PROGRAM main
VAR
	Relay_Start AT %QX4.0 : bool; (* Address modbus: 32 *)
	Start_State AT %QX4.1 : bool; (* Address modbus: 33 *)
	Relay_Downtime AT %QX4.2 : bool; (* Address modbus: 34 *)
	Downtime_State AT %QX4.3 : bool; (* Address modbus: 35 *)
	Counter_Trigger AT %QX4.4 : bool; (* Address modbus: 36 *)
	Reset_Counter AT %QX4.5 : bool; (* Address modbus: 37 *)
	Counter_Register AT %MW10 : int; (* 0 = 1024 --> HR 10 = 1034 *)
	R_TRIG0 : R_TRIG;
	Pulse_Counter : bool;
	CTU0 : CTU;
	R_TRIG1 : R_TRIG;
	Pulse_Reset : bool;
END_VAR

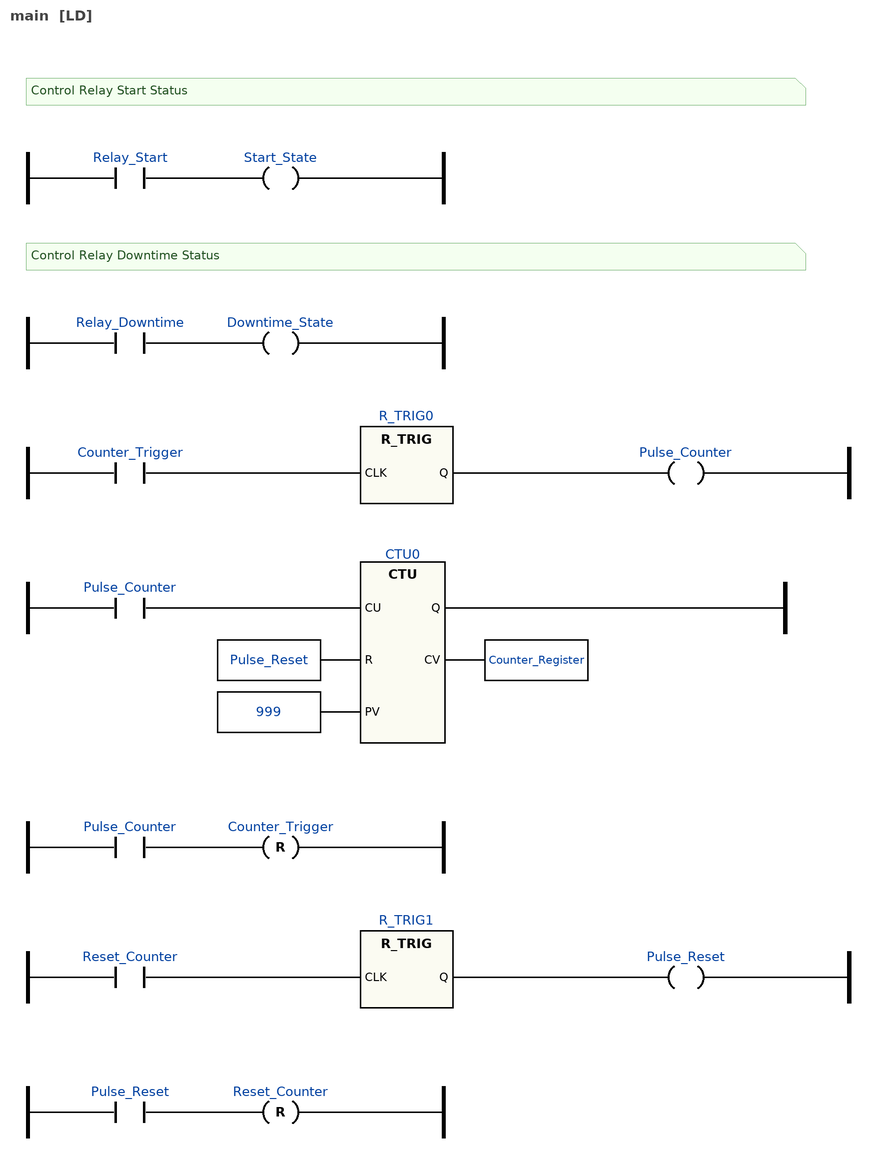
(* LD diagram, written out as Structured Text *)
(* Control Relay Start Status *)
Start_State := Relay_Start;
(* Control Relay Downtime Status *)
Downtime_State := Relay_Downtime;
R_TRIG0(CLK := Counter_Trigger);
Pulse_Counter := R_TRIG0.Q;
CTU0(CU := Pulse_Counter, R := Pulse_Reset, PV := 999);
Counter_Register := CTU0.CV;
IF Pulse_Counter THEN Counter_Trigger := FALSE; END_IF;
R_TRIG1(CLK := Reset_Counter);
Pulse_Reset := R_TRIG1.Q;
IF Pulse_Reset THEN Reset_Counter := FALSE; END_IF;
END_PROGRAM
